FUNCTION_BLOCK InfluentFeed_HMI (* Service Interface Function Block Type *)
  (* Standard: 61499-2 *)
  (* Version 0.0, 13/09/2026, template *)
  PACKAGE Hidryco.HidrycoLib;
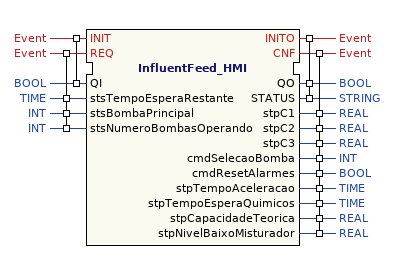
  EVENT_INPUT
    INIT WITH QI;
    REQ WITH stsTempoEsperaRestante, stsBombaPrincipal, stsNumeroBombasOperando;
  END_EVENT
  EVENT_OUTPUT
    INITO WITH QO, STATUS;
    CNF WITH stpC1, stpC2, stpC3, cmdSelecaoBomba, cmdResetAlarmes, stpTempoAceleracao, stpTempoEsperaQuimicos, stpCapacidadeTeorica, stpNivelBaixoMisturador;
  END_EVENT
  VAR_INPUT
    QI : BOOL;
    stsTempoEsperaRestante : TIME;
    stsBombaPrincipal : INT;
    stsNumeroBombasOperando : INT;
  END_VAR
  VAR_OUTPUT
    QO : BOOL; (* Event Output Qualifier *)
    STATUS : STRING; (* Service Status *)
    stpC1 : REAL; (* Gatilho para pedir a segunda bomba *)
    stpC2 : REAL; (* Evita degrau de vazão na partida *)
    stpC3 : REAL; (* Gatilho para tirar uma bomba *)
    cmdSelecaoBomba : INT;
    cmdResetAlarmes : BOOL;
    stpTempoAceleracao : TIME; (* Espera antes de controlar as duas bombas juntas *)
    stpTempoEsperaQuimicos : TIME; (* Espera para reiniciar após pH e condutividade normalizarem *)
    stpCapacidadeTeorica : REAL; (* Vazão nominal, para a malha aberta *)
    stpNivelBaixoMisturador : REAL; (* Bloqueio para misturadores *)
  END_VAR
  SERVICE /
    SEQUENCE 
    END_SEQUENCE
  END_SERVICE
END_FUNCTION_BLOCK
